DATA_BLOCK "CalcVolume_Tank9_DB"
{ S7_Optimized_Access := 'FALSE' }
VERSION : 0.1
"CalculationVolume"

BEGIN
   IW_Radius := 1.468;
   IW_ValueFromSensor := 18.20747;
   IW_K_for_Tonnag := 1.35;
   IW_K_for_Level := 1.35;
   QW_Volume := 91.26359;
   QW_Tonnag := 123.2058;
   QW_RealLevel := 13.48701;
   sW_S := 6.766776;
   sW_Volume := 91.26359;
   sW_RealLevel := 13.48701;

END_DATA_BLOCK

